Universal Robots URScript: EGH80_is_gripped_test.script

def EGH80_is_gripped_test():
  set_standard_analog_input_domain(0, 1)
  set_standard_analog_input_domain(1, 1)
  set_tool_analog_input_domain(0, 1)
  set_tool_analog_input_domain(1, 1)
  set_analog_outputdomain(0, 0)
  set_analog_outputdomain(1, 0)
  set_input_actions_to_default()
  set_tcp(p[0.0,0.0,0.23,0.0,0.0,0.0])
  set_payload(1.17, [-0.003, 0.002, 0.053])
  set_tool_communication(False, 115200, 0, 1, 1.5, 3.5)
  set_tool_output_mode(0)
  set_tool_digital_output_mode(0, 1)
  set_tool_digital_output_mode(1, 1)
  set_tool_voltage(0)
  step_count_b5384ae0_469d_4171_9f9b_4e9ab85c563a = 0.0
  thread Step_Counter_Thread_69980587_4d9a_4ef2_8bc1_6bf1d2362b1d():
    while (True):
      step_count_b5384ae0_469d_4171_9f9b_4e9ab85c563a = step_count_b5384ae0_469d_4171_9f9b_4e9ab85c563a + 1.0
      sync()
    end
  end
  run Step_Counter_Thread_69980587_4d9a_4ef2_8bc1_6bf1d2362b1d()
  set_gravity([0.0, 0.0, 9.82])
  set_safety_mode_transition_hardness(1)
  # begin: URCap Installation Node
  #   Source: DTI UR Library, 0.3.0, Danish Technological Institute
  #   Type: DTI UR Library
  ############################################################################
  # Copyright (C) Danish Technological Institute - All Rights Reserved       #
  # Unauthorized copying of this file, via any medium is strictly prohibited #
  # Proprietary and confidential                                             #
  # Written by Jens-Jakob Bentsen <jebe@dti.dk>, November 2020               #
  #                                                                          #
  # Force based moving and force checking                                    #
  #                                                                          #
  # Version                                                                  #
  dti_force_version = 2                                                      #
  #                                                                          #
  # dependencies on other DTI script files                                   #
  # int_dummy = NO_DEPENDENCIES                                              #
  #                                                                          #
  ############################################################################

  def get_dti_force_version():
    return dti_force_version
  end

  def get_dti_force_deps():
    # NO DEPS
    return True
  end


  # like UR's builtin get_tcp_force(), but return the force and torque values transformed
  # along the axes of the given pose
  # param pose: any valid pose, defaults to base, the x, y, and z values are ignored
  # return: 6D force vector with [Fx, Fy, Fz, Mx, My, Mz] aligned to pose in N and Nm respectively
  def get_tcp_force_in_frame(pose=p[0.0, 0.0, 0.0, 0.0, 0.0, 0.0]):

    # we are only interested in the rotation of pose, set translations to zero
    local target_pose = pose
    target_pose[0] = 0
    target_pose[1] = 0
    target_pose[2] = 0

    # the conversion needs to happen as poses, so we need to convert back and forth a bit
    local force = get_tcp_force()
    local force_vector_as_pose = p[force[0], force[1], force[2], 0, 0, 0]
    local torque_vector_as_pose = p[force[3], force[4], force[5], 0, 0, 0]
    local transformed_force_as_pose = pose_trans(pose_inv(target_pose), force_vector_as_pose)
    local transformed_torque_as_pose = pose_trans(pose_inv(target_pose),torque_vector_as_pose)
    return [transformed_force_as_pose[0], transformed_force_as_pose[1], transformed_force_as_pose[2], transformed_torque_as_pose[0], transformed_torque_as_pose[1], transformed_torque_as_pose[2]]
  end

  # get the force or torque values at the TCP along a single axis of the given pose
  # param axis: number of axis of pose, 0=x, 1=y, ...
  # param pose:  any valid pose, defaults to base, , the x, y, and z values are ignored
  # return: force or torque value in N or Nm respectively
  def get_tcp_force_1d(axis, pose=p[0.0, 0.0, 0.0, 0.0, 0.0, 0.0]):
    local force_vector = get_tcp_force_in_frame(pose)
    return force_vector[axis]
  end

  # perform a linear move while constantly checking the force; the move is aborted
  # if the force is exceeded and the robot is stopped
  # note: utilizes the currently active TCP
  # note: while running, check the value of the "current_force_vector" variable to check your forces in the given reference pose
  # param p_target: traget pose in base frame
  # param move_parameters: array [r, a, v] with
  #                        r: blend radius for linear move in m
  #                        a: accleration for linear move in m/s^2
  #                        v: velocity for linear move in m/s
  # param max_forces: maximum allowed absolute force in N along the reference pose's x, y, and z axis as vector [Fx, Fy, Fz]
  # param ignore_dists: array of [start_dist, end_dist] ignore the force value within these distances from the
  #                     start and end point, respectively
  #                     (gets around high force readings from acceleration / deceleration)
  # param refrence_pose: measure the allowed forces along the axes of this pose, defaults to the robot's base,
  #                      x, y, and z values of the pose are ignored
  # return: True if end of linear move was reached, else False
  def movel_checkforce(p_target, move_parameters, max_forces, ignore_dists=[0.0, 0.0], reference_pose=p[0.0, 0.0, 0.0, 0.0, 0.0, 0.0]):

    global p_thread_move_target = p_target
    global thread_move_params = move_parameters
    global thread_target_reached = False
    local p_current = get_actual_tcp_pose()  # current pose
    local p_start = get_actual_tcp_pose()  # start pose of move

    # we use this thread to do the moving
    thread move_thread():
      movel(p_thread_move_target, a=thread_move_params[0], v=thread_move_params[1], r=thread_move_params[2])
      thread_target_reached = True
      sync()
      sync()
    end

    # spin the moving thread and keep track of the force
    move_thread_handler = run move_thread()
    while(not thread_target_reached):
      p_current = get_actual_tcp_pose()
      global current_force_vector = get_tcp_force_in_frame(reference_pose)
      if point_dist(p_current, p_start) > ignore_dists[0] and point_dist(p_current, p_target) > ignore_dists[1]:
        if (norm(current_force_vector[0]) > max_forces[0]) or (norm(current_force_vector[1]) > max_forces[1]) or (norm(current_force_vector[2]) > max_forces[2]):
          kill move_thread_handler
          stopl(1)  # TODO: make this value accessible?
          return False
        end
      end
      sync()
    end
    return True
  end


  # Note 1 to self: a target pose in a feature can be converted to the robot's base frame by
  # using pose_in_base = pose_trans(feature_name, pose_in_feature)
  # end: URCap Installation Node
  # begin: URCap Installation Node
  #   Source: EGH-SCHUNK, 1.0.1, SCHUNK GmbH & Co. KG
  #   Type: SCHUNK EGH Gripper
    EGH = rpc_factory("xmlrpc", "http://127.0.0.1:40408/RPC2")
  global error_updated = False
  global error_internal = 0
  def EGH_error():
          if EGH.getActStatus() != 3:
              if error_updated == False:
                  error_internal = EGH.getDetailDeviceStatus(1)
                  error_updated = True
              end
              return error_internal
          else:
              error_updated = False
              error_internal = 0
              return 0
          end
  end
  def EGH_reference_ok():
          sync()
          return EGH.get_Referenced()
  end
  def EGH_is_success():
          sync()
          return EGH.isSuccess()
  end
  def EGH_is_blocked():
          sync()
          return EGH.isBlocked()
  end
  def EGH_is_endstop():
          sync()
          return EGH.isEndStop()
  end
  def EGH_is_closed():
          sync()
          return EGH.isClosed()
  end
  def EGH_is_open():
          sync()
          return EGH.isOpen()
  end
  def EGH_in_pos():
          sync()
          return EGH.isInPosition()
  end
  def EGH_actual_pos():
          sync()
          return EGH.get_CurrentPosition()
  end
  def EGH_status():
          sync()
          return EGH.getActStatus()
  end
  def EGH_error_check(name):
      local err =  EGH_status()
      if (err != 3):
          local err =  EGH_error()
          err_msg = EGH.getErrorMsg(err)
          textmsg(name, err_msg)
          popup(err_msg, title=name, error=True, blocking=True)
      end
      EGH_conn_check(name)
  end
  def EGH_conn_check(name):
      if (not EGH.is_connected()):
          err_msg = "Gripper disconnected"
          textmsg(name, err_msg)
          popup(err_msg, title=name, error=True, blocking=True)
          halt
      end
  end
  def EGH_goto_pos(value):
          sync()
      EGH.cmdPositioning(value)
  end
  def EGH_gripped_workpiece(wp):
      return EGH.isGrippedWp(wp)
  end

  EGH.resetPrgBreak()
  Gripper_LB_Enabled = True
  if (Gripper_LB_Enabled):
    set_digital_out(0, False)
    set_digital_out(1, True)
  end
  # end: URCap Installation Node
  def EGH80_connect():
    $ 6 "EGH80_connect" "noBreak"
    $ 7 "EGH.set_Ip('192.168.1.253')"
    EGH.set_Ip("192.168.1.253")
    $ 8 "EGH.connect( True )"
    EGH.connect(  True  )
    # begin: URCap Program Node
    #   Source: EGH-SCHUNK, 1.0.1, SCHUNK GmbH & Co. KG
    #   Type: EGH Color Light band
    $ 9 "EGH Color Light band "
    set_standard_digital_out(1, False)
    set_standard_digital_out(0, True)
    # end: URCap Program Node
    # begin: URCap Program Node
    #   Source: EGH-SCHUNK, 1.0.1, SCHUNK GmbH & Co. KG
    #   Type: EGH Commands
    $ 10 "EGH Acknowledge"
        EGH_conn_check("EGH Commands")
        EGH.cmdAcknowledge()
         while(EGH_status() == 0 ):
             EGH.cmdAcknowledge()
             sync()
         end
         sleep(0.200)
    # end: URCap Program Node
    # begin: URCap Program Node
    #   Source: EGH-SCHUNK, 1.0.1, SCHUNK GmbH & Co. KG
    #   Type: EGH Commands
    $ 11 "EGH Reference"
        EGH_error_check("EGH Commands")
        EGH.cmdReferencing()
         while(not EGH_reference_ok() and EGH_is_success() != True ):
        EGH_error_check("EGH Commands")
         end
    # end: URCap Program Node
    # begin: URCap Program Node
    #   Source: EGH-SCHUNK, 1.0.1, SCHUNK GmbH & Co. KG
    #   Type: EGH Commands
    $ 12 "EGH Acknowledge"
        EGH_conn_check("EGH Commands")
        EGH.cmdAcknowledge()
         while(EGH_status() == 0 ):
             EGH.cmdAcknowledge()
             sync()
         end
         sleep(0.200)
    # end: URCap Program Node
    # begin: URCap Program Node
    #   Source: EGH-SCHUNK, 1.0.1, SCHUNK GmbH & Co. KG
    #   Type: EGH Color Light band
    $ 13 "EGH Color Light band "
    Gripper_LB_Enabled=True
    set_standard_digital_out(1, True)
    set_standard_digital_out(0, False)
    # end: URCap Program Node
  end
  def EGH80_grip():
    $ 14 "EGH80_grip" "noBreak"
    # begin: URCap Program Node
    #   Source: EGH-SCHUNK, 1.0.1, SCHUNK GmbH & Co. KG
    #   Type: EGH Grip
    $ 15 "EGH Grip"
        EGH_error_check("EGH Grip")
        if(not EGH_reference_ok()):
            popup("Gripper not referenced", title="EGH Grip", error=True, blocking=True)
        else:
            EGH.set_DesiredPosition(16.14)
            sync()
            EGH.cmdGrip(0,0,0)
            while(EGH_is_success() != True and EGH_is_blocked() != True and EGH.isPrgBreak() == False):
                EGH_error_check("EGH Grip")
                sync()
            end
        end
    # end: URCap Program Node
    $ 16 "Wait: 1.5"
    sleep(1.5)
    $ 17 "If EGH_is_success()≟ True  and EGH_is_endstop()≠ True "
    if ( EGH_is_success () ==   True    and   EGH_is_endstop () !=   True  ):
      # begin: URCap Program Node
      #   Source: EGH-SCHUNK, 1.0.1, SCHUNK GmbH & Co. KG
      #   Type: EGH Color Light band
      $ 18 "EGH Color Light band "
      Gripper_LB_Enabled=True
      set_standard_digital_out(1, True)
      set_standard_digital_out(0, False)
      # end: URCap Program Node
      $ 19 "return True "
      return  True
    else:
      $ 20 "Else" "noBreak"
      # begin: URCap Program Node
      #   Source: EGH-SCHUNK, 1.0.1, SCHUNK GmbH & Co. KG
      #   Type: EGH Color Light band
      $ 21 "EGH Color Light band "
      set_standard_digital_out(1, True)
      set_standard_digital_out(0, True)
      # end: URCap Program Node
      $ 22 "return  False "
      return   False
    end
  end
  $ 1 "BeforeStart"
  $ 2 "Call EGH80_connect"
  EGH80_connect()
  $ 3 "Robot Program"
  # begin: URCap Program Node
  #   Source: EGH-SCHUNK, 1.0.1, SCHUNK GmbH & Co. KG
  #   Type: EGH Grip
  $ 4 "EGH Release"
      EGH_error_check("EGH Grip")
      if(not EGH_reference_ok()):
          popup("Gripper not referenced", title="EGH Grip", error=True, blocking=True)
      else:
          EGH.cmdRelease(0)
          while(EGH_is_success() != True and EGH_is_blocked() != True and EGH.isPrgBreak() == False):
              EGH_error_check("EGH Grip")
              sync()
          end
      end
  # end: URCap Program Node
  $ 5 "is_gripped≔EGH80_grip()"
  global is_gripped=EGH80_grip()
end
